(* IEC 61131-3 sources: Std_PalletMover/Class/CntrlPeriperalPiviotWheels, 1 file *)

(* ---- CntrlPeriperalPiviotWheels.st ---- *)
(*!
<Class
	Name               = "CntrlPeriperalPiviotWheels"
	Revision           = "0.0"
	RealtimeTask       = "false"
	CyclicTask         = "false"
	BackgroundTask     = "false"
	Sigmatek           = "false"
	OSInterface        = "false"
	HighPriority       = "false"
	Automatic          = "false"
	UpdateMode         = "Prescan"
	SharedCommandTable = "true"
	Objectsize         = "(750,120)">
	<Channels>
		<Client Name="ToAgvConfig" Required="true" Internal="false"/>
		<Client Name="ToAgvSettings" Required="true" Internal="false"/>
	</Channels>
	<Network Name="CntrlPeriperalPiviotWheels">
		<!-- List of Components in this network -->
		<Components>
			<Object
				Name       = "_base"
				Class      = "PeripheralsBase"
				Position   = "(218,120)"
				Visualized = "false">
				<Channels>
					<Server Name="ObjectStatus"/>
					<Server Name="ToObject"/>
					<Client Name="op_LogData"/>
					<Client Name="p_NextObject"/>
				</Channels>
			</Object>
		</Components>
		<Comments>
		</Comments>
		<!-- List of Connections in this network -->
		<Connections>
			<Connection Source="this.ToObject" Destination="_base.ToObject" Vertices="(976,210),(804,210),"/>
			<Connection Source="_base.p_NextObject" Destination="this.p_NextObject" Vertices="(218,270),(38,270),"/>
			<Connection Source="_base.op_LogData" Destination="this.op_LogData" Vertices="(218,210),(38,210),"/>
		</Connections>
		<!-- Headerfiles -->
		<Options>
		</Options>
	</Network>
</Class>
*)
#pragma using PeripheralsBase

CntrlPeriperalPiviotWheels : CLASS
: PeripheralsBase
  //Servers:
  //Clients:
	ToAgvConfig 	: CltChCmd_AgvConfig;
	ToAgvSettings 	: CltChCmd_AgvSettings;
  //Variables:
  //Functions:
  //Tables:
	FUNCTION @STD
		VAR_OUTPUT
			ret_code	: CONFSTATES;
		END_VAR;
	FUNCTION GLOBAL TAB @CT_;
END_CLASS;

#pragma usingLtd AgvConfig
#pragma usingLtd AgvSettings
